PROGRAM MAIN
VAR
END_VAR

TcUnit.RUN();

END_PROGRAM

(* stored: Version 1.1.0.1, ProductVersion 3.1.4024.15
   POU MAIN: Id {1c7dbdb3-3ad9-058e-2a75-807bd1bcee45}, SpecialFunc None *)
